(* IEC 61131-3 sources: Industry-PLC-LLM/data/PLCBEAD_repo/PLCBEAD_PLCEmbed-main/PLC-BEAD/Source/GEB/FIFO_32, 1 file *)

(* ---- FIFO_32.ST ---- *)
TYPE
	oscat_ardw_0_31             : ARRAY [0..31]   OF DWORD;
END_TYPE

FUNCTION INC1:INT

	VAR_INPUT
		X :	INT;
		N :	INT;
	END_VAR

	IF X >= N - 1 THEN
		INC1 := 0;
	ELSE
		INC1 := X + 1;
	END_IF;
END_FUNCTION

FUNCTION_BLOCK FIFO_32

	VAR_INPUT
		DIN :	DWORD;
		E :	BOOL := TRUE;
		RD :	BOOL;
		WD :	BOOL;
		RST :	BOOL;
	END_VAR

	VAR_OUTPUT
		DOUT :	DWORD;
		EMPTY :	BOOL := TRUE;
		FULL :	BOOL;
	END_VAR

	VAR
		fifo :	oscat_ardw_0_31;
		pr :	INT;
		pw :	INT;
	END_VAR

	IF RST THEN
		pw := pr;
		FULL := FALSE;
		EMPTY := TRUE;
		DOUT := DWORD#0;
	ELSIF E THEN
		IF NOT EMPTY AND RD THEN
			DOUT := fifo[pr];
			pr := INC1(pr,32);
			EMPTY := pr = pw;
			FULL := FALSE;
		END_IF;
		IF NOT FULL AND WD THEN
			fifo[pw] := DIN;
			pw := INC1(pw,32);
			FULL := pw = pr;
			EMPTY := FALSE;
		END_IF;
	END_IF;

END_FUNCTION_BLOCK

PROGRAM program0
  VAR
	DIN :	DWORD;
	E   :	BOOL;
	RD  :	BOOL;
	WD  :	BOOL;
	RST :	BOOL;

	DOUT  :	DWORD;
	EMPTY :	BOOL;
	FULL  :	BOOL;

	func_block : FIFO_32;
  END_VAR
	func_block.DIN :=DIN;
	func_block.E   :=E  ;
	func_block.RD  :=RD ;
	func_block.WD  :=WD ;
	func_block.RST :=RST;
	func_block();
	DOUT := func_block.DOUT ;
	EMPTY:= func_block.EMPTY;
	FULL := func_block.FULL ;
END_PROGRAM
